FUNCTION_BLOCK COURIER_DISCOVERY (* Composite Function Block Type *)
  (* Standard: 61499-2 *)
  (* Version 0.0, 12/17/2022, Dmitrii, Flexbridge AB, template *)
  PACKAGE UAO.Hackathon;
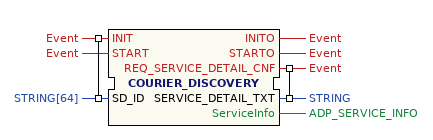
  EVENT_INPUT
    INIT WITH SD_ID;
    START;
  END_EVENT
  EVENT_OUTPUT
    INITO;
    STARTO;
    REQ_SERVICE_DETAIL_CNF WITH SERVICE_DETAIL_TXT;
  END_EVENT
  VAR_INPUT
    SD_ID : STRING[64];
  END_VAR
  VAR_OUTPUT
    SERVICE_DETAIL_TXT : STRING;
  END_VAR
  PLUGS
    ServiceInfo : ADP_SERVICE_INFO;
  END_PLUGS
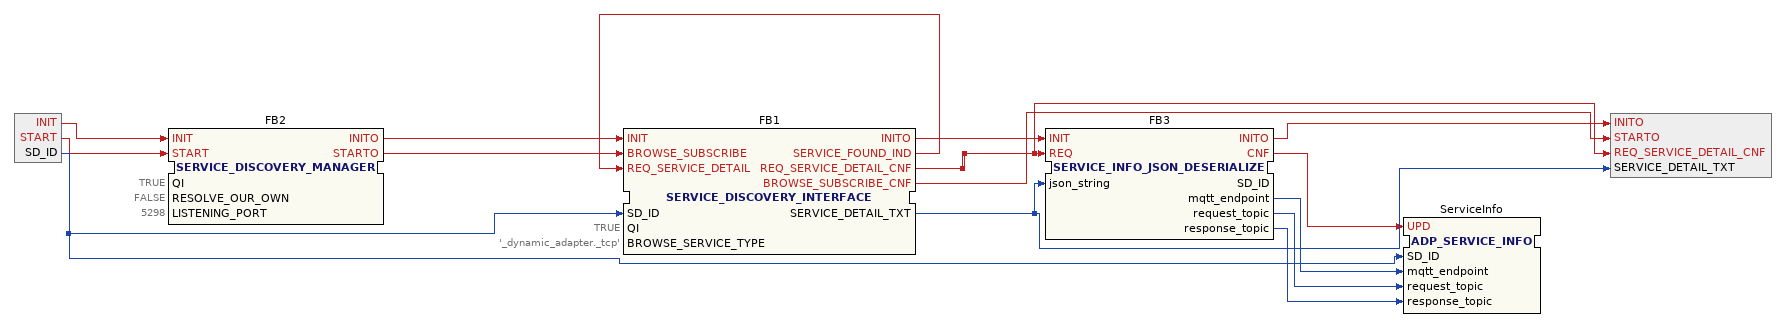
  FBS
    FB1 : SERVICE_DISCOVERY_INTERFACE(QI := TRUE, BROWSE_SERVICE_TYPE := '_dynamic_adapter._tcp');
    FB2 : SERVICE_DISCOVERY_MANAGER(QI := TRUE, RESOLVE_OUR_OWN := FALSE, LISTENING_PORT := 5298);
    FB3 : SERVICE_INFO_JSON_DESERIALIZE;
  END_FBS
  EVENT_CONNECTIONS
    INIT TO FB2.INIT;
    FB2.INITO TO FB1.INIT;
    FB1.INITO TO FB3.INIT;
    FB3.CNF TO ServiceInfo.UPD;
    FB2.STARTO TO FB1.BROWSE_SUBSCRIBE;
    FB1.SERVICE_FOUND_IND TO FB1.REQ_SERVICE_DETAIL;
    FB1.REQ_SERVICE_DETAIL_CNF TO FB3.REQ;
    FB3.INITO TO INITO;
    FB1.BROWSE_SUBSCRIBE_CNF TO STARTO;
    START TO FB2.START;
    FB1.REQ_SERVICE_DETAIL_CNF TO REQ_SERVICE_DETAIL_CNF;
  END_CONNECTIONS
  DATA_CONNECTIONS
    SD_ID TO ServiceInfo.SD_ID;
    FB1.SERVICE_DETAIL_TXT TO FB3.json_string;
    FB3.mqtt_endpoint TO ServiceInfo.mqtt_endpoint;
    FB3.request_topic TO ServiceInfo.request_topic;
    FB3.response_topic TO ServiceInfo.response_topic;
    SD_ID TO FB1.SD_ID;
    FB1.SERVICE_DETAIL_TXT TO SERVICE_DETAIL_TXT;
  END_CONNECTIONS
END_FUNCTION_BLOCK
